FUNCTION_BLOCK OR_2 (* FB to calculate bitwise boolean OR (generic FB) *)
  {SET_ATTRIBUTE(eclipse4diac::core::GenericClassName, 'GEN_OR')}
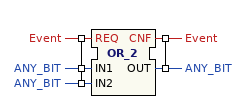
  EVENT_INPUT
    REQ WITH IN1, IN2; (* Normal Execution Request *)
  END_EVENT
  EVENT_OUTPUT
    CNF WITH OUT; (* Execution Confirmation *)
  END_EVENT
  VAR_INPUT
    IN1 : ANY_BIT; (* OR input 1 *)
    IN2 : ANY_BIT; (* OR input 2 *)
  END_VAR
  VAR_OUTPUT
    OUT : ANY_BIT; (* OR result *)
  END_VAR
END_FUNCTION_BLOCK
